FUNCTION_BLOCK FB_Blink_S
VAR_INPUT
	Tv:TIME;		(*Czas trwania impulsu i przerwy*)
END_VAR
VAR_OUTPUT
	Q:BOOL;			(*Wyjscie*)
END_VAR
VAR
	ton1: TON;
END_VAR

ton1(IN:= TRUE, PT:= 2*Tv, Q=> , ET=> );
Q := ton1.ET > Tv;
IF ton1.Q THEN
	ton1(IN:= FALSE);
END_IF

END_FUNCTION_BLOCK

(* stored: Version 1.1.0.1, ProductVersion 3.1.4022.12
   POU FB_Blink_S: Id {cf256ac7-7962-4767-9504-b3ad334176c8}, SpecialFunc None *)
